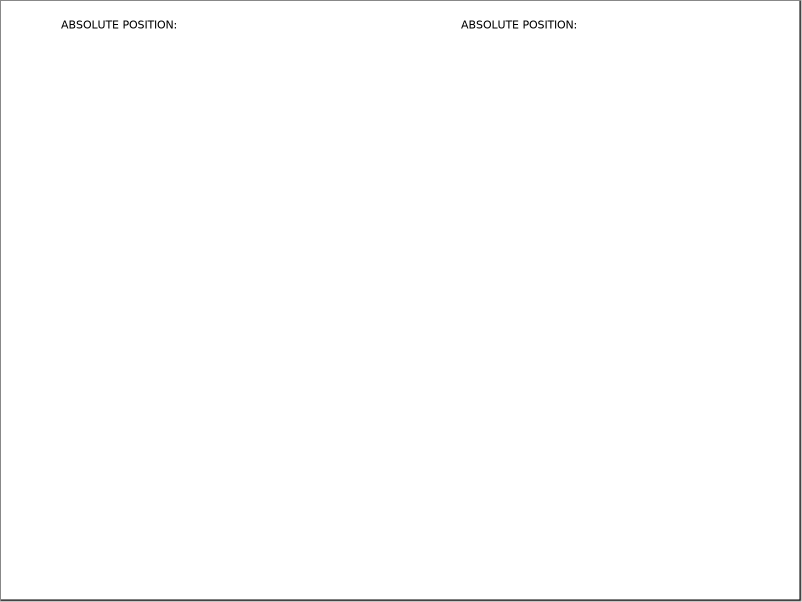
VISUALIZATION F27_Halt  // 802x602
    Rectangle (0,0 800x600)
    Label (10,10 170x30), "ABSOLUTE POSITION:"
    Label (410,10 170x30), "ABSOLUTE POSITION:"
END_VISUALIZATION

(* stored: Version 1.1.0.1, ProductVersion 3.1.4022.7
   Visu F27_Halt: Id {ebb8f23d-4a5b-4736-b994-bb8193b9128b} *)
